PROGRAM PRG_TEST
VAR
	HeatingCurve_Test : FC_HeatingCurve_Test;							 
END_VAR

TcUnit.RUN();

END_PROGRAM

(* stored: Version 1.1.0.1, ProductVersion 3.1.4024.6
   POU PRG_TEST: Id {152e68d5-965f-4c54-a511-098a773e86b5}, SpecialFunc None *)
